Fanuc KAREL source: ks00055.KL

PROGRAM KS00055
%STACKSIZE=65535
%PRIORITY=65535
%NOLOCKGROUP
VAR
FLAG : BOOLEAN
N : INTEGER
STATUS : INTEGER
PN : STRING[80]
VN : STRING[80]
-- UNRESOLVED DECLARATIONS (source type spelling not recovered)
-- A : ARRAY[4] OF TYPE_0x1100 (type_u16=0x3100)
-- B : ARRAY[4] OF TYPE_0x1100 (type_u16=0x3100)
BEGIN
PN=''
VN='A'
-- UNRESOLVED_PC line 19 opcodes [27 22 22 2A 22 2A 22 22 AF] marker_code=27
END KS00055
